PROGRAM MAIN
VAR
END_VAR

END_PROGRAM

(* stored: Version 1.1.0.1
   POU MAIN: Id {ea66bf43-71f2-4ef8-987d-6506258bd22c} *)
